// Setup can legitimately be slow. It must not spend the body's scan budget doing

// it, or a fixture waiting on hardware would time out work that never started.

//

// A body budget of ONE, and a setup taking four scans. If the two shared a clock

// this test would report a timeout instead of a pass.
FUNCTION_BLOCK TEST_RunnerSetupDoesNotSpendTheBodyBudget IMPLEMENTS I_Test
VAR
	// A private runner, driven one scan per call. The outer test spans scans by

	// returning FALSE, which is exactly the mechanism being verified one level down.
	Registry	   : TestRegistry<1>;
	Runner		   : TestRunner;
	Handle		   : TestVerdict;
	Budgets		   : ST_TestBudgets;
	Journal		   : REFERENCE TO TestJournal;
	Slot		   : ST_TestSlot;
	Outcome		   : E_PhaseOutcome;
	Loaded		   : BOOL;
	Phase		   : DINT;
	Scans		   : DINT;
	Subject		   : SlowSetupTest;
	ExpectedZero   : UDINT;
	ExpectedFour   : UDINT;
	ExpectedOne	   : UDINT;
	ActualCount	   : UDINT;
	ExpectedStatus : E_TestStatus;
	ActualStatus   : E_TestStatus;
END_VAR

METHOD Run : BOOL
VAR_INPUT
	Enable : BOOL;
	Test   : I_TestAssertions;
END_VAR
Scans := Scans + 1;
IF Scans > 200 THEN
	Test.Fail('the subject never reached a terminal outcome');
	Run := TRUE;
	RETURN;
END_IF

CASE Phase OF
	0:
		// One scan for the body. Four for setup, from the suite default, which is
		// deliberately left disabled here so setup cannot expire.
		Budgets.Body.Cycles		 := 1;
		Budgets.Body.IsCyclesSet := TRUE;
		Registry.TryClaim(Subject, 'slow setup', Budgets);
		Runner.Attach(Roster := Registry, Verdict := Handle);
		Slot   := Registry.Slot(0);
		Loaded := Runner.Load(Slot);
		Phase  := 1;
		Run	   := FALSE;

	1:
		Outcome := Runner.Advance(Enable := TRUE);
		IF Outcome <> E_PhaseOutcome.Running THEN
			Phase := 2;
		END_IF

		Run := FALSE;

	2:
		ExpectedFour := 4;
		ActualCount	 := Subject.SetupCalls;
		Test.AssertEqual(ExpectedFour, ActualCount, 'setup took four scans');
		ExpectedOne := 1;
		ActualCount := Subject.BodyCalls;
		Test.AssertEqual(ExpectedOne, ActualCount, 'the body still got its scan');

		// The proof: had setup spent the body budget, this would be four.
		ExpectedZero := 0;
		ActualCount	 := Subject.CyclesAtStart;
		Test.AssertEqual(ExpectedZero, ActualCount, 'the body started at zero cycles');
		Test.AssertTrue(Subject.FirstCycleAtStart, 'and its first call was the first cycle');
		Journal REF= Registry.Journal(0);
		IF __ISVALIDREF(Journal) THEN
			ExpectedStatus := E_TestStatus.Passed;
			ActualStatus   := Journal.Status;
			Test.AssertEqual(ExpectedStatus, ActualStatus, 'passed, not timed out');
		END_IF

		Run := TRUE;
END_CASE
END_METHOD

END_FUNCTION_BLOCK

(* stored: Version 1.1.0.1, ProductVersion 3.1.4026.18
   POU TEST_RunnerSetupDoesNotSpendTheBodyBudget: Id {03a568b3-f78a-4298-a177-a05052841d05}, SpecialFunc None
   Folder I_Test: Id {fd885154-af25-42dd-bea5-28c03de44830}
   Method Run: Id {e0201a95-6c65-4d8e-b712-6d8258f087b9} *)
